FUNCTION_BLOCK ABSTRACT SuspendedToReadyProgramTransition EXTENDS ProgramTransition

{attribute 'monitoring' := 'call'}
{attribute 'OPC.UA.DA.Property' := '1'}
{attribute 'OPC.UA.DA.Access' := '1'}
PROPERTY FINAL Cause : STRING
GET
Cause := 'Reset';
END_GET
END_PROPERTY

{attribute 'monitoring' := 'call'}
{attribute 'OPC.UA.DA.Property' := '1'}
{attribute 'OPC.UA.DA.Access' := '1'}
PROPERTY FINAL FromState : STRING
GET
FromState := 'Suspended';
END_GET
END_PROPERTY

{attribute 'monitoring' := 'call'}
{attribute 'OPC.UA.DA.Property' := '1'}
{attribute 'OPC.UA.DA.Access' := '1'}
PROPERTY FINAL Name : STRING
GET
Name := 'SuspendedToReady';
END_GET
END_PROPERTY

{attribute 'monitoring' := 'call'}
{attribute 'OPC.UA.DA.Property' := '1'}
{attribute 'OPC.UA.DA.Access' := '1'}
PROPERTY FINAL ToState : STRING
GET
ToState := 'Ready';
END_GET
END_PROPERTY

END_FUNCTION_BLOCK

(* stored: Version 1.1.0.1
   POU SuspendedToReadyProgramTransition: Id {dc74d145-21a0-4551-9761-225af06dd512}, SpecialFunc None
   Property Cause: Id {d4acb4ef-a083-4cfd-bd16-672ecc6b1b22}
   Get Get: Id {952b5430-3c5a-4073-b6be-7809ca8a6ef3}
   Property FromState: Id {a4344b52-65f8-48af-a16f-3568d81b72d0}
   Get Get: Id {54c7a6e2-a226-48bb-81ef-f85153058fe4}
   Property Name: Id {36209df9-4a93-4223-9823-60c827646282}
   Get Get: Id {be7d2b31-d759-4c8c-b077-285414ba23f7}
   Property ToState: Id {b3c7346d-e5d4-4fd1-9a26-79f624325f4e}
   Get Get: Id {ede6727f-1bf6-497c-b811-771d313243fb} *)
